# EPICS autosave request: ipApp/Db/XIA_pfcu_filters_settings.req
$(P)$(F):filter1_thick
$(P)$(F):filter2_thick
$(P)$(F):filter3_thick
$(P)$(F):filter4_thick
$(P)$(F):filter1_thick.EGU
$(P)$(F):filter2_thick.EGU
$(P)$(F):filter3_thick.EGU
$(P)$(F):filter4_thick.EGU
$(P)$(F):filter1_mat
$(P)$(F):filter2_mat
$(P)$(F):filter3_mat
$(P)$(F):filter4_mat
$(P)$(F):filter1_other
$(P)$(F):filter2_other
$(P)$(F):filter3_other
$(P)$(F):filter4_other
